# EPICS autosave request: iocBoot/gmca_23o_ioc1/dbSave/BP_Mo_.req
%
% BURT Request File
%
% $(P)BP:Mo:  BPM after DCM
%

file assy.req ASSY=$(P)BP:Mo
file mtr1.req MTR1=$(P)BP:mmo
file drv1.req DRV1=$(P)BP:MOZ
